PROGRAM PLC_PRG
VAR


END_VAR

END_PROGRAM
